PROGRAM FB_KJL300
VAR
	AO:INT;
	rPRESS:REAL;
	xPRESS_OK:BOOL;
	xHV_DIS:BOOL:=TRUE;
END_VAR

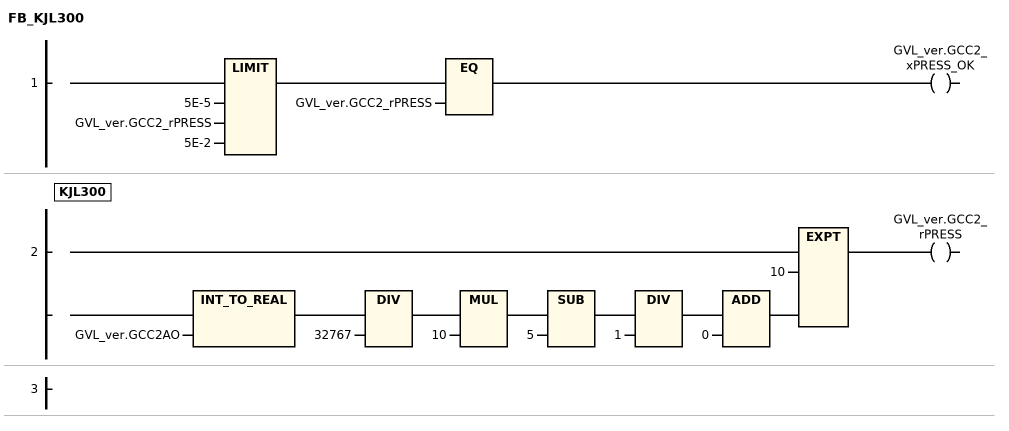
// NETWORK 1
GVL_ver.GCC2_xPRESS_OK := LIMIT(5E-5, GVL_ver.GCC2_rPRESS, 5E-2) = GVL_ver.GCC2_rPRESS;

// NETWORK 2
KJL300:
GVL_ver.GCC2_rPRESS := EXPT(10, ((INT_TO_REAL(GVL_ver.GCC2AO) / 32767) * 10 - 5) / 1 + 0);

// NETWORK 3

END_PROGRAM

(* stored: Version 1.1.0.1, ProductVersion 3.1.4022.3
   POU FB_KJL300: Id {03e84ac8-8255-4ff2-9f53-b59d3dc04968}, SpecialFunc None *)
